// TIA Portal V17 export
// export: Created 2024-09-02T12:49:55.4510922Z, ExportSetting WithDefaults, DisplayName Totally Integrated Automation Portal, DisplayVersion V17, DisplayName TIA Portal Openness, DisplayVersion V17, DisplayName TIA Portal Version Control Interface, DisplayVersion V17, DisplayName STEP 7 Professional, DisplayVersion V17, DisplayName STEP 7 Safety, DisplayVersion V17, DisplayName WinCC Professional, DisplayVersion V17
FUNCTION "SysFC_HMI_ScreenCall" : Void   // FC258, LAD
TITLE = Select screen / Bildanwahl
{ S7_Optimized_Access := 'TRUE' }
AUTHOR : OlegFuehrus
FAMILY : HMI
NAME : HMI
VERSION : 1.0
// stored: AutoNumber true, IsIECCheckEnabled false, SetENOAutomatically false, UDAEnableTagReadback false
   VAR_INPUT
      i_Start : Bool;   // Start des Bildaufrufes / Start of the screen call
      i_ScreenNr : Int;   // Bildnummer / Screen number
   END_VAR
   VAR_IN_OUT
      io_LTLL_Data : "LTLL_typeData";   // Bereichszeiger / Area pointer
   END_VAR
   VAR_TEMP
      t_ScreenNr : Int;
      t_ScreenActive : Bool;
   END_VAR
BEGIN

REGION Network 1: Current screen number read / aktuelle Bildnummer lesen
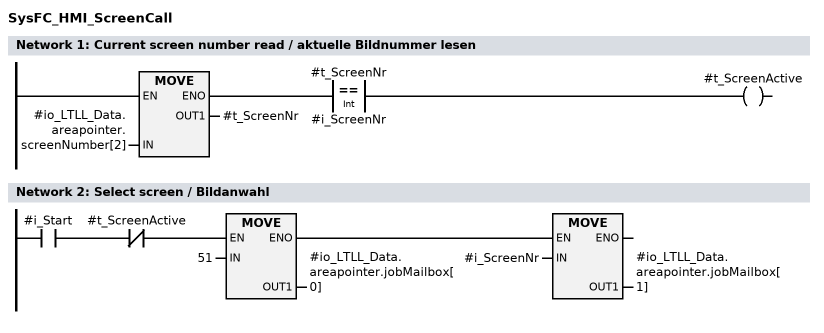
   RUNG wire#powerrail
      Move(in := #io_LTLL_Data.areapointer.screenNumber[2], out1 => #t_ScreenNr)
      { S7_Templates := "SrcType := Int" } EQ_Contact(in1 := #t_ScreenNr, in2 := #i_ScreenNr)
      Coil( #t_ScreenActive )
   END_RUNG
   // the same network as SCL:
   #t_ScreenNr := #io_LTLL_Data.areapointer.screenNumber[2];
   #t_ScreenActive := #t_ScreenNr = #i_ScreenNr;
END_REGION

REGION Network 2: Select screen / Bildanwahl
   RUNG wire#powerrail
      Contact( #i_Start )
      I_Contact( #t_ScreenActive )
      Move(in := 51, out1 => #io_LTLL_Data.areapointer.jobMailbox[0])
      Move(in := #i_ScreenNr, out1 => #io_LTLL_Data.areapointer.jobMailbox[1])
   END_RUNG
   // the same network as SCL:
   IF #i_Start AND NOT #t_ScreenActive THEN
       #io_LTLL_Data.areapointer.jobMailbox[0] := 51;
       #io_LTLL_Data.areapointer.jobMailbox[1] := #i_ScreenNr;
   END_IF;
END_REGION
END_FUNCTION
